// Mitsubishi GX Works2 project: 传数值的另一种写法2   PLC: L02S

FUNCTION_BLOCK xsz
VAR_INPUT
  IN1 : BOOL;
END_VAR
VAR_OUTPUT
  OUT1 : BOOL;
END_VAR
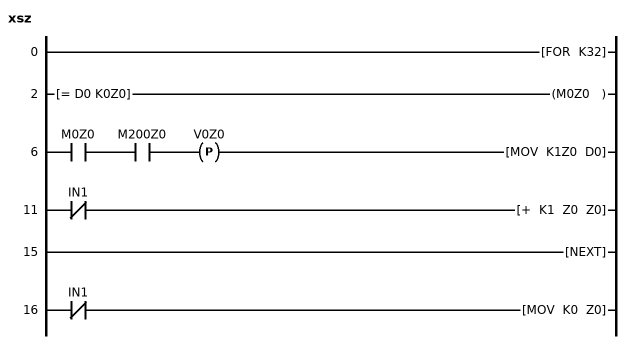
0     FOR     K32
2     LD=     D0 K0Z0
      OUT     M0Z0
6     LD      M0Z0
      AND     M200Z0
      EGP     V0Z0
      MOV     K1Z0 D0
11    LDI     IN1
      +       K1 Z0 Z0
15    NEXT
16    LDI     IN1
      MOV     K0 Z0
END_FUNCTION_BLOCK

PROGRAM xszxsz
VAR
  xsz_1 : xsz;
END_VAR
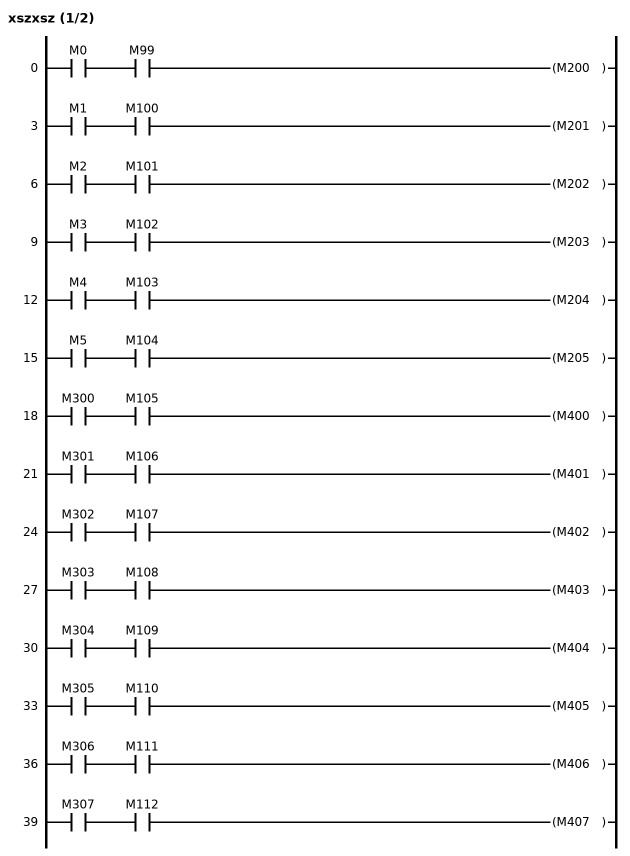
0     LD      M0
      AND     M99
      OUT     M200
3     LD      M1
      AND     M100
      OUT     M201
6     LD      M2
      AND     M101
      OUT     M202
9     LD      M3
      AND     M102
      OUT     M203
12    LD      M4
      AND     M103
      OUT     M204
15    LD      M5
      AND     M104
      OUT     M205
18    LD      M300
      AND     M105
      OUT     M400
21    LD      M301
      AND     M106
      OUT     M401
24    LD      M302
      AND     M107
      OUT     M402
27    LD      M303
      AND     M108
      OUT     M403
30    LD      M304
      AND     M109
      OUT     M404
33    LD      M305
      AND     M110
      OUT     M405
36    LD      M306
      AND     M111
      OUT     M406
39    LD      M307
      AND     M112
      OUT     M407
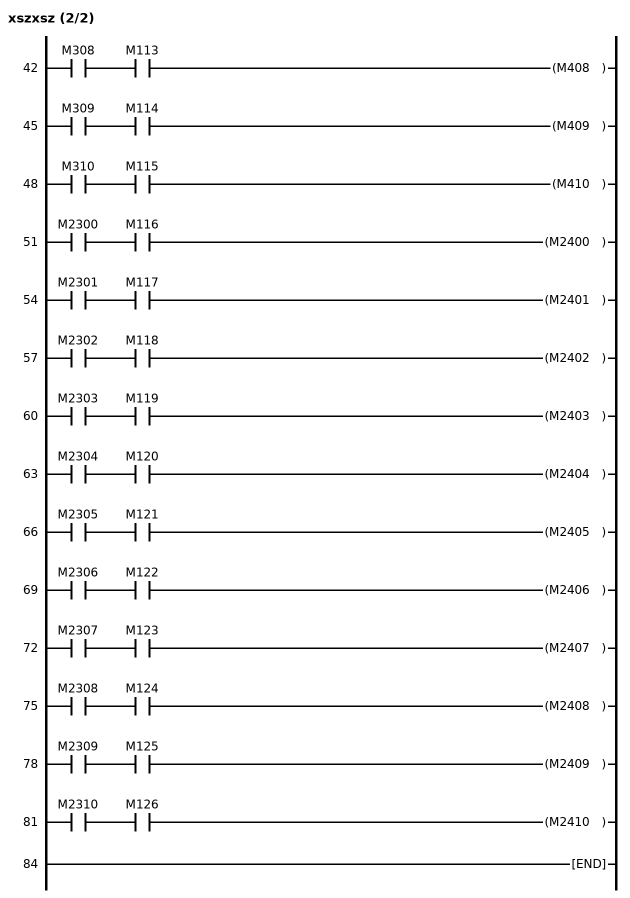
42    LD      M308
      AND     M113
      OUT     M408
45    LD      M309
      AND     M114
      OUT     M409
48    LD      M310
      AND     M115
      OUT     M410
51    LD      M2300
      AND     M116
      OUT     M2400
54    LD      M2301
      AND     M117
      OUT     M2401
57    LD      M2302
      AND     M118
      OUT     M2402
60    LD      M2303
      AND     M119
      OUT     M2403
63    LD      M2304
      AND     M120
      OUT     M2404
66    LD      M2305
      AND     M121
      OUT     M2405
69    LD      M2306
      AND     M122
      OUT     M2406
72    LD      M2307
      AND     M123
      OUT     M2407
75    LD      M2308
      AND     M124
      OUT     M2408
78    LD      M2309
      AND     M125
      OUT     M2409
81    LD      M2310
      AND     M126
      OUT     M2410
84    END
END_PROGRAM

PROGRAM aas
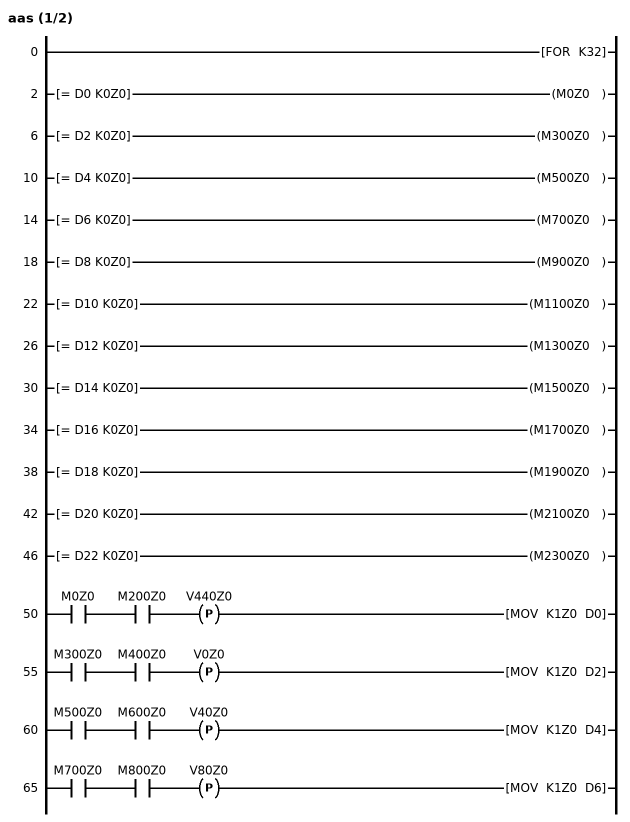
0     FOR     K32
2     LD=     D0 K0Z0
      OUT     M0Z0
6     LD=     D2 K0Z0
      OUT     M300Z0
10    LD=     D4 K0Z0
      OUT     M500Z0
14    LD=     D6 K0Z0
      OUT     M700Z0
18    LD=     D8 K0Z0
      OUT     M900Z0
22    LD=     D10 K0Z0
      OUT     M1100Z0
26    LD=     D12 K0Z0
      OUT     M1300Z0
30    LD=     D14 K0Z0
      OUT     M1500Z0
34    LD=     D16 K0Z0
      OUT     M1700Z0
38    LD=     D18 K0Z0
      OUT     M1900Z0
42    LD=     D20 K0Z0
      OUT     M2100Z0
46    LD=     D22 K0Z0
      OUT     M2300Z0
50    LD      M0Z0
      AND     M200Z0
      EGP     V440Z0
      MOV     K1Z0 D0
55    LD      M300Z0
      AND     M400Z0
      EGP     V0Z0
      MOV     K1Z0 D2
60    LD      M500Z0
      AND     M600Z0
      EGP     V40Z0
      MOV     K1Z0 D4
65    LD      M700Z0
      AND     M800Z0
      EGP     V80Z0
      MOV     K1Z0 D6
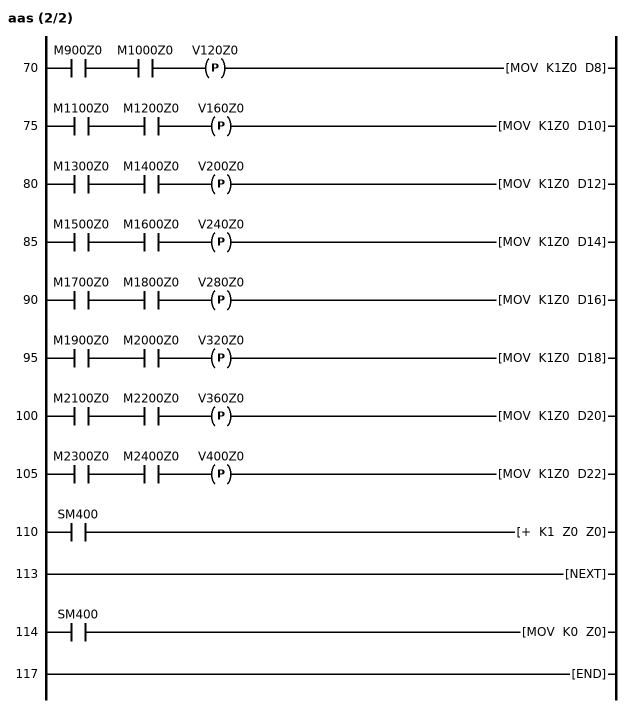
70    LD      M900Z0
      AND     M1000Z0
      EGP     V120Z0
      MOV     K1Z0 D8
75    LD      M1100Z0
      AND     M1200Z0
      EGP     V160Z0
      MOV     K1Z0 D10
80    LD      M1300Z0
      AND     M1400Z0
      EGP     V200Z0
      MOV     K1Z0 D12
85    LD      M1500Z0
      AND     M1600Z0
      EGP     V240Z0
      MOV     K1Z0 D14
90    LD      M1700Z0
      AND     M1800Z0
      EGP     V280Z0
      MOV     K1Z0 D16
95    LD      M1900Z0
      AND     M2000Z0
      EGP     V320Z0
      MOV     K1Z0 D18
100   LD      M2100Z0
      AND     M2200Z0
      EGP     V360Z0
      MOV     K1Z0 D20
105   LD      M2300Z0
      AND     M2400Z0
      EGP     V400Z0
      MOV     K1Z0 D22
110   LD      SM400
      +       K1 Z0 Z0
113   NEXT
114   LD      SM400
      MOV     K0 Z0
117   END
END_PROGRAM
